{attribute 'pack_mode' := '1'}
TYPE ST_EncoderSample:
STRUCT
    extTime	: T_DCTIME64; (* The time of the sample. Beckhoff TAI-like external time.*)
    pos		: LREAL; (* Axis position in mm. *)
END_STRUCT
END_TYPE

(* stored: Version 1.1.0.1, ProductVersion 3.1.4022.18
   DUT ST_EncoderSample: Id {9977e928-4a64-437c-9c03-77e732264d83} *)
